{attribute 'qualified_only'}
{attribute 'strict'}
TYPE EFeedbackMsgAttenuationELL14k :
(
	StateMsg := 1,
	PositionMsg := 10,
    IdMsg,
    CustomMsg
);
END_TYPE

(* stored: Version 1.1.0.1, ProductVersion 3.1.4024.4
   DUT EFeedbackMsgAttenuationELL14k: Id {8ba5a620-346a-4159-8bea-d9cc79f74a04} *)
